FUNCTION_BLOCK FB_Math
VAR_INPUT
END_VAR
VAR_OUTPUT
END_VAR
VAR
END_VAR

METHOD AddTwo : REAL
VAR_INPUT
	Real1 :REAL;
	Real2 :REAL;
END_VAR

AddTwo := Real1 + Real2;
AddTwo := Real1 + Real2;
AddTwo := Real1 + Real2;
AddTwo := Real1 + Real2;
AddTwo := Real1 + Real2;
END_METHOD

END_FUNCTION_BLOCK

(* stored: Version 1.1.0.1, ProductVersion 3.1.4022.18
   POU FB_Math: Id {6fbab0f8-a7af-456d-8d51-f26ee1045dbf}, SpecialFunc None
   Method AddTwo: Id {7197c489-6d7a-4f1e-8c2b-9cccebb0429f} *)
